{attribute addProperty BoxType "EL9222-4433-0018"}
{attribute addProperty Id "StatusAT %I*Status_EBB67327324"}
{attribute addProperty CRC "4261982012"}
{attribute addProperty SizeInBites "32"}
{attribute addProperty SizeInBytes "4"}
TYPE OCP_Inputs_Channel_FE08AF3C :
STRUCT
	{attribute addProperty Name "Status"}
	Status AT %I* : Status_EBB67327;
END_STRUCT
END_TYPE

(* stored: Version 1.2.0.0, ProductVersion 3.1.4024.9
   DUT OCP_Inputs_Channel_FE08AF3C: Id {24408ca5-8b80-4014-b8ba-09af61f2e9cf} *)
